(* CODESYS project Pult.project

Project tree, tasks and I/O mapping:
  Device : Owen SPK1xx, Owen, order no. 023, version 3.5.4.20
    application Application
      libraries: Standard, * (System); CAA SerialCom, 3.5.5.0 (CAA Technical Workgroup); CAA Types Extern, 3.5.5.0 (CAA Technical Workgroup); VisuDialogs, * (System); Standard64, * (System); ModBus, 3.2.0 (OWEN); ComSerice, 3.1.0 (OWEN); SysCom, 3.5.5.0 (System)
      task MainTask (cyclic, interval t#10ms, priority 1) calls PLC_PRG
      task VISU_TASK (cyclic, interval 100 ms, priority 31) calls VisuElems.Visu_Prg
      program PLC_PRG [ST]: acDelay
      visualisation main
    Modbus_COM : Modbus COM, 3S - Smart Software Solutions GmbH, version 3.4.0.0 (disabled)
        settings: DataBits = 8; StopBits = 1; ComPort = 2
      Modbus_Serial_Device : Modbus Serial Device, 3S - Smart Software Solutions GmbH, version 3.5.5.0
          unmapped channels: Inputs, Outputs
  libraries: CAA SerialCom, 3.5.5.0 (CAA Technical Workgroup); CAA Types Extern, 3.5.5.0 (CAA Technical Workgroup)
  ComPortFB/
    function block ComPortFB [ST]: mInit, mRead, mStopRead, mWrite
    data type ComPortSettingsST
    ENUMs/
      data type ComParityENUM
      data type ComNumberENUM
      data type ComBaudrateENUM
      data type ComStopBitsENUM
    global variables ComPortFB_GVL_Constant
  text list GlobalTextList
  ModbusFB_v1.0/
    function block ModbusFB [ST]: mReadMV110_16, mWriteMU110_8, mReadMV110_8A, mInitModbus, mWrite16, mRead03, mRead04
    data type FunctionMBE
    data type ReadingRegistrValueST
    global variables GVL_ModbusConstant
*)

// ComPortFB/ComPortSettingsST
TYPE ComPortSettingsSt :
STRUCT
	ComPortN: ComNumberENUM;
	Baudrate: ComBaudrateENUM;
	Parity: ComParityENUM;
	StopBits: COMStopBitsENUM;
	tTimeOut: TIME;	//таймаут ответа
END_STRUCT
END_TYPE

// ComPortFB/ENUMs/ComParityENUM
TYPE ComParityENUM :
(
	COM_NONE_PARITY := 0,
	COM_ODD_PARITY,
	COM_EVEN_PARITY
);
END_TYPE

// ComPortFB/ENUMs/ComNumberENUM
TYPE ComNumberENUM :
(
	COM_N1 := 1,
	COM_N2,
	COM_N3,
	COM_N4,
	COM_N5
);
END_TYPE

// ComPortFB/ENUMs/ComBaudrateENUM
TYPE ComBaudrateENUM :
(
	COM_BAUDRATE_4800,
	COM_BAUDRATE_9600,
	COM_BAUDRATE_19200,
	COM_BAUDRATE_38400,
	COM_BAUDRATE_57600,
	COM_BAUDRATE_115200,
	COM_BAUDRATE_230400,
	COM_BAUDRATE_460800,
	COM_BAUDRATE_921600
);
END_TYPE

// ComPortFB/ENUMs/ComStopBitsENUM
TYPE ComStopBitsENUM :
(
	COM_ONE_BITS := 0,
	COM_TWO_BITS
);
END_TYPE

// ModbusFB_v1.0/FunctionMBE
TYPE FunctionMBE :
(
	MBNoneFun,	//нет функции
	MBwrite,	//функция modbus 16
	MBread		//функция modbus 03
);
END_TYPE

// ModbusFB_v1.0/ReadingRegistrValueST
TYPE ReadingRegistrValueST :
STRUCT
	wMV110_16: WORD;
	arwMV110_8A: ARRAY[1..8] OF WORD;
	arwRead03: ARRAY[1..ModbusMaxArraySize] OF WORD;
	arwRead04: ARRAY[1..ModbusMaxArraySize] OF WORD;
END_STRUCT
END_TYPE

// ComPortFB/ComPortFB_GVL_Constant
VAR_GLOBAL CONSTANT
	iMaxByteQty: INT:=255;
END_VAR

// ModbusFB_v1.0/GVL_ModbusConstant
VAR_GLOBAL CONSTANT
	ModbusMaxArraySize: BYTE:=100;	// - максимальное количество опрашиваемых за раз регистров WORD
END_VAR

// Device/Application/PLC_PRG
PROGRAM PLC_PRG
VAR
	bInit: BOOL;
	fbCOM: ComPortFB;
	stCOMSettings: ComPortSettingsSt;
	TON1: TON;
	ar: ARRAY[0..iMaxByteQty] OF BYTE;
	byPWM: BYTE;
	byFreqHi: BYTE;	//точно
	byFreqLo: BYTE;	//грубо
	byPWMBack: BYTE;
	byFreqHiBack: BYTE;	//точно
	byFreqLoBack: BYTE;	//грубо	
	bWrite: BOOL;
	arRead: ARRAY[0..2] OF BYTE;
	ADC1: WORD;
	ADC2: WORD;
	wsFreq: WSTRING;
	
	oMB: ModbusFB;
	iSt: INT;
	arwBuf: ARRAY[1..ModbusMaxArraySize] OF WORD;		//буфер для функций отправки
	bIndOn: BOOL;
	bLightBack: BOOL;
END_VAR
VAR_TEMP
	wTemp: WORD;
END_VAR

IF NOT(bInit) THEN
	oMB.stSettings.byParity:=SYS_NOPARITY;
	oMB.stSettings.byStopBits:=SysCom.SYS_ONESTOPBIT;
	oMB.stSettings.sPort:=SysCom.SYS_COMPORT2;
	oMB.stSettings.ulBaudrate:=SysCom.SYS_BR_9600;
	oMB.stSettings.ulTimeout:=SYS_NOWAIT;
	oMB.stSettings.ulBufferSize:=0;
	bInit:=oMB.mInitModbus();
ELSE
	CASE iSt OF
		0: 
			IF oMB.mRead03(16#0A,0,2) THEN
				IF NOT(oMB.bError) THEN
					ADC1:=oMB.RegistrValue.arwRead03[1];
					ADC2:=oMB.RegistrValue.arwRead03[2];
				END_IF	
				iSt:=iSt+1;	
			END_IF
		1:
			acDelay();
		2:
			iSt:=0;
	END_CASE
END_IF

ACTION acDelay:
			TON1(IN:=TRUE,PT:=T#10MS);
			IF TON1.Q THEN
				TON1(IN:=FALSE);
				iSt:=iSt+1;
			END_IF
END_ACTION

END_PROGRAM

// ComPortFB/ComPortFB
FUNCTION_BLOCK ComPortFB	//ФБ работы ком порта без протокола
VAR_INPUT
END_VAR
VAR_OUTPUT
	wsState: WSTRING;		//строка состояния
	bError: BOOL;			//флаг ошибки
	arReadData: ARRAY[0..iMaxByteQty] OF BYTE;			//принятые данные
	iQtyRead: UINT;		//количество принятых mRead байтов
END_VAR
VAR
	fbOpen: COM.Open;		//фб открытия
	fbWrite: COM.Write;		//фб отправки
	fbRead: COM.Read;		//фб приёма
	bOpen: BOOL;			//флаг открытия
	Handle: CAA.HANDLE;		//инициализатор
	InitStep: INT;			//служебная mInit
	WriteStep: INT;			//служебная mWrite
	ReadStep: INT;			//служебная mRead
	arComParams : ARRAY [1..7] OF COM.PARAMETER;	//для инициализации
	arBuf: ARRAY[0..iMaxByteQty] OF BYTE;			//буффер
	TONTimeOut: TON;
	tTimeOut: TIME;
END_VAR

;

METHOD mInit : BOOL //инициализация порта (одновременно его открытие)
VAR_INPUT
	stCOMSettings: ComPortSettingsSt;
END_VAR
VAR
END_VAR
IF NOT(bOpen) THEN
	mInit:=FALSE;
	IF stCOMSettings.tTimeOut=T#0S THEN
		tTimeOut:=T#100MS;
	ELSE
		tTimeOut:=stCOMSettings.tTimeOut;
	END_IF
	CASE InitStep OF
		0:	arComParams[1].udiParameterId:=COM.CAA_Parameter_Constants.udiPort;
			arComParams[1].udiValue:=INT_TO_UINT(stCOMSettings.ComPortN);
			arComParams[2].udiParameterId:=COM.CAA_Parameter_Constants.udiBaudrate;
			CASE stCOMSettings.Baudrate OF
				ComBaudrateENUM.COM_BAUDRATE_4800: arComParams[2].udiValue:=4800;
				ComBaudrateENUM.COM_BAUDRATE_9600: arComParams[2].udiValue:=9600;
				ComBaudrateENUM.COM_BAUDRATE_19200: arComParams[2].udiValue:=19200;
				ComBaudrateENUM.COM_BAUDRATE_38400: arComParams[2].udiValue:=38400;
				ComBaudrateENUM.COM_BAUDRATE_57600: arComParams[2].udiValue:=57600;
				ComBaudrateENUM.COM_BAUDRATE_115200: arComParams[2].udiValue:=115200;
				ComBaudrateENUM.COM_BAUDRATE_230400: arComParams[2].udiValue:=230400;
				ComBaudrateENUM.COM_BAUDRATE_460800: arComParams[2].udiValue:=460800;
				ComBaudrateENUM.COM_BAUDRATE_921600: arComParams[2].udiValue:=921600;
			END_CASE
			arComParams[3].udiParameterId:=COM.CAA_Parameter_Constants.udiParity;
			CASE stCOMSettings.Parity OF
				ComParityENUM.COM_NONE_PARITY: arComParams[3].udiValue:=INT_TO_UDINT(COM.PARITY.NONE);
				ComParityENUM.COM_ODD_PARITY: arComParams[3].udiValue:=INT_TO_UDINT(COM.PARITY.ODD);
				ComParityENUM.COM_EVEN_PARITY: arComParams[3].udiValue:=INT_TO_UDINT(COM.PARITY.EVEN);
			END_CASE
			arComParams[4].udiParameterId:=COM.CAA_Parameter_Constants.udiStopBits;
			CASE stCOMSettings.StopBits OF
				ComStopBitsENUM.COM_ONE_BITS: arComParams[4].udiValue:=INT_TO_UDINT(COM.STOPBIT.ONESTOPBIT);
				ComStopBitsENUM.COM_TWO_BITS: arComParams[4].udiValue:=INT_TO_UDINT(COM.STOPBIT.TWOSTOPBITS);
			END_CASE
			arComParams[5].udiParameterId:=COM.CAA_Parameter_Constants.udiByteSize;
			arComParams[5].udiValue:=8;
			arComParams[6].udiParameterId:=COM.CAA_Parameter_Constants.udiTimeout;
			arComParams[6].udiValue:=0;
			arComParams[7].udiParameterId:=COM.CAA_Parameter_Constants.udiBinary;
			arComParams[7].udiValue:=0;
			fbOpen.usiListLength:=INT_TO_USINT(SIZEOF(arComParams));
			fbOpen.pParameterList:=ADR(arComParams);
			fbOpen(xExecute:=FALSE);
			InitStep:=InitStep+1;
		1:	fbOpen(xExecute:=TRUE);
			IF fbOpen.xDone THEN
				bOpen:=TRUE;
				wsState:="Порт открыт";
				InitStep:=0;
				bError:=FALSE;
				Handle:=fbOpen.hCom;
			END_IF
			IF fbOpen.xError THEN
				wsState:="Ошибка открытия";
				bError:=TRUE;
				InitStep:=0;
			END_IF
	END_CASE//CASE InitStep OF
ELSE//IF NOT(bOpen) THEN
	InitStep:=0;
	mInit:=TRUE;
END_IF
END_METHOD

METHOD mRead: BOOL
VAR_INPUT
	iByteQty: UINT;
END_VAR
VAR
	i : INT;
END_VAR
IF bOpen THEN
	CASE ReadStep OF
		0:	//обнуление выходного массива
			FOR i:=0 TO iMaxByteQty DO
				arReadData[i]:=0;
			END_FOR
			fbRead(xExecute:=FALSE);
			ReadStep:=ReadStep+1;
			iQtyRead:=0;
			bError:=FALSE;
			TONTimeOut(IN:=FALSE);
		1:	TONTimeOut(IN:=TRUE,PT:=tTimeOut);
			fbRead.xExecute:=TRUE;
			fbRead.hCom:=Handle;
			fbRead.pBuffer:=ADR(arReadData);
			fbRead.szBuffer:=(*CAA.UINT_TO_SIZE*)(iByteQty);
			fbRead();
			iQtyRead:=CAA.SIZE_TO_UINT(fbRead.szSize);
			IF fbRead.xError THEN
				bError:=TRUE;
				wsState:="Ошибка приёма";
				ReadStep:=0;
			ELSIF TONTimeOut.Q THEN
				bError:=TRUE;
				wsState:="Ошибка таймаута";
				ReadStep:=0;
			ELSIF iQtyRead=iByteQty THEN
				bError:=FALSE;
				wsState:="Принято";
				ReadStep:=0;
				mRead:=TRUE;
			END_IF
	END_CASE
ELSE//IF bOpen THEN
	wsState:="Порт не открыт";
	bError:=TRUE;
END_IF
END_METHOD

METHOD mStopRead	//останавливает приём данных
VAR_INPUT
END_VAR
bError:=FALSE;
wsState:="Приём остановлен";
ReadStep:=0;
END_METHOD

METHOD mWrite : BOOL	//отправляет iByteQty байт из массива arData, возвращает true по завершению
VAR_INPUT
	arData: ARRAY[0..iMaxByteQty] OF BYTE;
	iByteQty: INT;
END_VAR
IF bOpen THEN
	CASE WriteStep OF
		0:	arBuf:=arData;
			fbWrite(xExecute:=FALSE);
			WriteStep:=WriteStep+1;
			bError:=FALSE;
		1:	fbWrite.xExecute:=TRUE;
			fbWrite.hCom:=Handle;
			fbWrite.pBuffer:=ADR(arBuf);
			fbWrite.szSize:=INT_TO_UDINT(iByteQty);
			fbWrite();
			IF fbWrite.xError THEN
				bError:=TRUE;
				wsState:="Ошибка отправки";
				WriteStep:=0;
			END_IF
			IF fbWrite.xDone THEN
				bError:=FALSE;
				wsState:="Отправлено";
				WriteStep:=0;
				mWrite:=TRUE;
			END_IF
	END_CASE
ELSE//IF bOpen THEN
	wsState:="Порт не открыт";
	bError:=TRUE;
END_IF
END_METHOD

END_FUNCTION_BLOCK

// ModbusFB_v1.0/ModbusFB
//должны быть добавлены следующие библиотеки
//	SysCom 3.5.5.0
//	ComSerice 3.1.0
//	ModBus 3.2.0
//должна быть создана глобальная константа ModbusArraySize - максимальное количество опрашиваемых за раз регистров WORD
FUNCTION_BLOCK ModbusFB
VAR_INPUT
	stSettings: COM_Settings;						//установки ком порта
END_VAR
VAR_OUTPUT
	ErrorCount: DWORD;		//счетчик ошибок
	bDone: BOOL;			//флаг выполненого обмена
	bError: BOOL;			//флаг ошибки (данные не обновлены)
	RegistrValue: ReadingRegistrValueST;
END_VAR
VAR
//	Adress: ENUMModbusAdr;	// адресов устройства
//	RegistrNum: BYTE;		// регистр, скоторого опрашивать
//	RegistQty: BYTE(1..ModbusMaxArraySize);		// количество регистров для чтения/записи
	RegistrIn: ARRAY[1..ModbusMaxArraySize] OF WORD;		// значение регистра для записи
//	MBFunction: ENUMFunctionMB;	//функция modbus
	bOpenPort: BOOL;
	COM_SERVICE1: COM_SERVICE; 		(*для открытия порта*)
	MB_16: MB_WR_REGS;				(*ФБ modbus функция 16 -  запись параметров (несколько регистров через буфер) *)
	MB_03: MB_RD_HOLD_REGS;			(*ФБ modbus функция 03 -  чтение параметров (несколько регистров через буфер) *)
	MB_04: MB_RD_INP_REGS;			(*ФБ modbus функция 04 -  чтение параметров (несколько регистров через буфер) *)
	Buffer: 		ARRAY[0..255] OF BYTE ; 
	Time_out:		TIME		:=T#200MS;	(*таймаут ответа*)
	RegistrOut: ARRAY[1..ModbusMaxArraySize] OF WORD;		//значение регистра после чтения
END_VAR
VAR_TEMP
	i: INT;
END_VAR

;

METHOD mReadMV110_16 : BOOL
VAR_INPUT
	Adress: INT;
END_VAR
mReadMV110_16:=FALSE;
IF mRead03(Adress,51,1) THEN
	mReadMV110_16:=TRUE;
	RegistrValue.wMV110_16:=RegistrValue.arwRead03[1];	
END_IF
END_METHOD

METHOD mWriteMU110_8 : BOOL
VAR_INPUT
	Adress: INT;
	Value: WORD;
END_VAR
RegistrIn[1]:=Value;
mWriteMU110_8:=mWrite16(Adress,50,RegistrIn,1);
END_METHOD

METHOD mReadMV110_8A : BOOL
VAR_INPUT
	Adress: INT;
	QtyIn: BYTE;			//количество подключенных датчиков (чтоб не опрашивать лишнее)
END_VAR
VAR
	i: INT;
END_VAR
mReadMV110_8A:=mRead03(Adress,1,(QtyIn-1)*6+1);
IF mReadMV110_8A THEN
	FOR i:=1 TO QtyIn DO
		RegistrValue.arwMV110_8A[i]:=RegistrValue.arwRead03[(i-1)*6+1];	
	END_FOR
END_IF
END_METHOD

METHOD mInitModbus : BOOL
VAR_INPUT
END_VAR
(*StSettings.byParity:=SYS_NOPARITY;
StSettings.byStopBits:=SYS_ONESTOPBIT;
StSettings.sPort:=SYS_COMPORT3;
StSettings.ulBaudrate:=SYS_BR_115200;
StSettings.ulTimeout:=SYS_NOWAIT;
*)
(*открываем COM порт*)
COM_SERVICE1(Enable:=NOT(bOpenPort),Settings:=StSettings,Task:=OPEN_TSK );	
bOpenPort:=COM_SERVICE1.ready;
mInitModbus:=bOpenPort;
END_METHOD

METHOD mWrite16 : BOOL
VAR_INPUT
	Adress:INT;
	FirstRegistrAdress: BYTE;
	WhatWrite: ARRAY[1..ModbusMaxArraySize] OF WORD;
	QtyWriteRegistr: BYTE(1..ModbusMaxArraySize);
END_VAR
VAR
	i: INT;
END_VAR
mWrite16:=FALSE;
bDone:=FALSE;
bError:=FALSE;

IF NOT(MB_16.Enable) THEN
	FOR i:=1 TO QtyWriteRegistr DO
		Buffer[2*i-1]:=WORD_TO_BYTE(WhatWrite[i]);
		Buffer[2*i-2]:=WORD_TO_BYTE(WhatWrite[i]/256);	
	END_FOR
END_IF

MB_16	(Enable:=TRUE,				
		Mode:=MB_RTU,				
		DevAddr:=INT_TO_BYTE(Adress),								
		FirstAddr:=FirstRegistrAdress, 				
		Quantity:=QtyWriteRegistr,   			
		Buffer:=Buffer,			
		ComHandle:=COM_SERVICE1.Handle,	
		TimeOut:=Time_out,			
	 	);
		
IF MB_16.Complete  THEN
	IF MB_16.Exception<>0 THEN
		ErrorCount:=ErrorCount+1;
		IF ErrorCount=1 THEN
			ErrorCount:=0;
			bDone:=TRUE;
			bError:=TRUE;
		END_IF
	ELSE								
		bDone:=TRUE;
		ErrorCount:=0;
	END_IF;
	MB_16(Enable:=FALSE,Buffer:=Buffer);
END_IF

IF bDone THEN
	mWrite16:=TRUE;
END_IF
END_METHOD

METHOD mRead03 : BOOL
VAR_INPUT
	Adress:INT;
	FirstRegistrAdress: BYTE;
	QtyWriteRegistr: BYTE(1..ModbusMaxArraySize);
END_VAR
VAR
	i: INT;
END_VAR
mRead03:=FALSE;
bDone:=FALSE;
bError:=FALSE;

MB_03	(Enable:=TRUE,					
		Mode:=MB_RTU,				
		DevAddr:=INT_TO_BYTE(Adress),					
		FirstAddr:=FirstRegistrAdress,					
		Quantity:=QtyWriteRegistr,			
		ComHandle:=COM_SERVICE1.Handle, 	
		TimeOut:=Time_out,
		Buffer:=Buffer,					
		);
		
IF MB_03.Complete AND MB_03.Exception<>0 THEN
	ErrorCount:=ErrorCount+1;
	IF ErrorCount=1 THEN
		ErrorCount:=0;
		bDone:=TRUE;
		bError:=TRUE;
	END_IF
END_IF

IF MB_03.Complete AND MB_03.Exception=0 THEN	
	FOR i:=1 TO QtyWriteRegistr DO
		RegistrOut[i]:=BYTE_TO_WORD(BUFFER[2*i-1]) OR SHL(BYTE_TO_WORD(BUFFER[2*i-2]),8);
	END_FOR
	bDone:=TRUE;
	ErrorCount:=0;
END_IF

IF bDone THEN
	mRead03:=TRUE;
	RegistrValue.arwRead03:=RegistrOut;
END_IF
END_METHOD

METHOD mRead04 : BOOL
VAR_INPUT
	Adress:INT;
	FirstRegistrAdress: BYTE;
	QtyWriteRegistr: BYTE(1..ModbusMaxArraySize);
END_VAR
VAR
	i: INT;
END_VAR
mRead04:=FALSE;
bDone:=FALSE;
bError:=FALSE;

MB_04	(Enable:=TRUE,					
		Mode:=MB_RTU,				
		DevAddr:=INT_TO_BYTE(Adress),					
		FirstAddr:=FirstRegistrAdress,					
		Quantity:=QtyWriteRegistr,			
		ComHandle:=COM_SERVICE1.Handle, 	
		TimeOut:=Time_out,
		Buffer:=Buffer,					
		);
		
IF MB_04.Complete AND MB_04.Exception<>0 THEN
	ErrorCount:=ErrorCount+1;
	IF ErrorCount=3 THEN
		ErrorCount:=0;
		bDone:=TRUE;
		bError:=TRUE;
	END_IF
END_IF

IF MB_04.Complete AND MB_04.Exception=0 THEN	
	FOR i:=1 TO QtyWriteRegistr DO
		RegistrOut[i]:=BYTE_TO_WORD(BUFFER[2*i-1]) OR SHL(BYTE_TO_WORD(BUFFER[2*i-2]),8);
	END_FOR
	bDone:=TRUE;
	ErrorCount:=0;
END_IF

IF bDone THEN
	mRead04:=TRUE;
	RegistrValue.arwRead04:=RegistrOut;
END_IF
END_METHOD

END_FUNCTION_BLOCK

// Device/Application/main
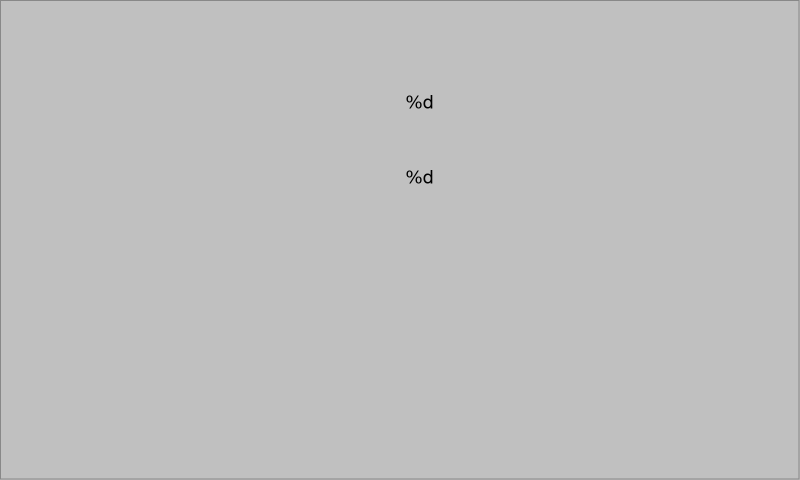
VISUALIZATION main  // 800x480
    Rectangle (340,80 160x45), "%d", text variable: PLC_PRG.ADC1
    Rectangle (340,155 160x45), "%d", text variable: PLC_PRG.ADC2
END_VISUALIZATION
